TYPE (* A Template for an Attribute Type *)
  (* Version 0.0, 2023-11-21, 4DIAC-IDE *)
END_TYPE
